// TwinCAT 3 PLC project Tc3_Event
// Title: Tc3_Event
// Company: www.peterzerlauth.com
// Author: Peter Zerlauth
// ProjectVersion: 0.0.0.7
// Description: Tc3_Event – TwinCAT 3 Event Logging Framework Copyright (c) Peter Zerlauth This component is provided under a Dual Licensing Model: 1. GPLv3 Open-Source License - Free for personal, educational, and non-commercial use. - Commercial use allowed only if the entire application is published under GPLv3, including all modifications to this code. - Requires full disclosure of source code for derivative works. 2. Commercial License - Required for integration into proprietary or closed-source products. - Removes all GPLv3 copyleft obligations. - Includes optional warranty, professional support, and long-term maintenance options. For commercial licensing, contact: info@peterzerlauth.com By using this Function Block you agree to the terms of the selected license.
// ProgramVersion: 3.1.4026.20
// libraries:
//   SysDir, * (System)
//   SysFile, * (System)
//   Tc2_Standard, * (Beckhoff Automation GmbH)
//   Tc2_System, * (Beckhoff Automation GmbH)
//   Tc2_Utilities, * (Beckhoff Automation GmbH)
//   Tc3_EventLogger, * (Beckhoff Automation GmbH)
//   Tc3_Module, * (Beckhoff Automation GmbH)
// project tree:
//   Argument/ FB_Argument.TcPOU (not stored), I_Argument.TcIO (not stored)
//   Event/ I_Event.TcIO, FB_Event.TcPOU
//   Global Variables/ GVL.TcGVL (not stored)
//   Helpers/File/ E_FileState.TcDUT (not stored), FB_File.TcPOU (not stored), I_File.TcIO (not stored)
//   Helpers/ F_Filter.TcPOU (not stored), F_Hash.TcPOU (not stored), F_InstancePath.TcPOU (not stored), F_Log.TcPOU (not stored), F_Print.TcPOU (not stored), F_Remove.TcPOU (not stored), LogLevel_To_Severity.TcPOU (not stored)
//   Logger/ E_LogLevel.TcDUT (not stored), I_Logger.TcIO (not stored)
//   Logger/FileLogger/ FB_FileLogger.TcPOU (not stored)
//   Logger/HmiLogger/ FB_HmiLogger.TcPOU (not stored)
//   Logger/Manager/ FB_LoggerManager.TcPOU (not stored)
//   Logger/TcLogger/ FB_TcLogger.TcPOU (not stored)
//   Message/ FB_Message.TcPOU (not stored)
//   Project Information/ F_GetCompany.TcPOU (not stored), F_GetTitle.TcPOU (not stored), F_GetVersion.TcPOU
//   Version/ Global_Version.TcGVL
// (motion and I/O tree: see PLC project plc01)
// real-time tasks:
//   TASK SlowTask: cycle T#20ms, priority 20, ADS port 350
//   TASK FastTask: cycle T#1ms, priority 1, ADS port 351

// ---- Version/Global_Version.TcGVL
{attribute 'TcGenerated'}
{attribute 'no-analysis'}
{attribute 'linkalways'}
// This function has been automatically generated from the project information.
VAR_GLOBAL CONSTANT
	{attribute 'const_non_replaced'}
	stLibVersion_Tc3_Event : ST_LibVersion := (iMajor := 0, iMinor := 0, iBuild := 0, iRevision := 7, nFlags := 0, sVersion := '0.0.0.7');
END_VAR

// ---- Event/I_Event.TcIO
INTERFACE I_Event

METHOD PUBLIC M_Critical : BOOL
VAR_INPUT
	sMessage:			STRING(255);
	nID:				UDINT;
END_VAR
END_METHOD

METHOD PUBLIC M_Error : BOOL
VAR_INPUT
	sMessage:			STRING(255);
	nID:				UDINT;
END_VAR
END_METHOD

METHOD PUBLIC M_Info : BOOL
VAR_INPUT
	sMessage:			STRING(255);
	nID:				UDINT;
END_VAR
END_METHOD

METHOD M_Reset : BOOL
VAR_INPUT
END_VAR
END_METHOD

METHOD PUBLIC M_Verbose : BOOL
VAR_INPUT
	sMessage:			STRING(255);
END_VAR
END_METHOD

METHOD PUBLIC M_Warning : BOOL
VAR_INPUT
	sMessage:			STRING(255);
	nID:				UDINT;
END_VAR
END_METHOD

PROPERTY PUBLIC P_Argument : I_Argument
GET
END_GET
END_PROPERTY

PROPERTY PUBLIC P_Logger : I_Logger
GET
END_GET
SET
END_SET
END_PROPERTY

END_INTERFACE

// ---- Event/FB_Event.TcPOU

{attribute 'reflection'} 
// Providing the event logger
FUNCTION_BLOCK FB_Event IMPLEMENTS I_Event
VAR_INPUT
	iLogger:					I_Logger;		// Interface has to be attached to a Valid target
END_VAR
VAR
    {attribute 'hide'} 
    {attribute 'instance-path'} 
    {attribute 'noinit'} 
    sInstancePath:				STRING(255);
	fbSymbolInfo: 				PLC_ReadSymInfoByNameEx;
	fbSystemTime: 				FB_LocalSystemTime;
	fbArguments:				FB_Argument;	
	fbVerbose:					FB_Message;
	fbInfo:						FB_Message;
	fbWarning:					FB_Message;
	fbError:					FB_Message;
	fbCritical:					FB_Message;
END_VAR
VAR_STAT
	nCycleTime:					UDINT;
	nTimestamp:					Tc2_Utilities.T_FILETIME64;		
END_VAR
(*
    Tc3_Event – TwinCAT 3 Event Logging Framework
    Copyright (c) Peter Zerlauth

    This component is provided under a Dual Licensing Model:

    1. GPLv3 Open-Source License
       - Free for personal, educational, and non-commercial use.
       - Commercial use allowed only if the entire application is published
         under GPLv3, including all modifications to this code.
       - Requires full disclosure of source code for derivative works.

    2. Commercial License
       - Required for integration into proprietary or closed-source products.
       - Removes all GPLv3 copyleft obligations.
       - Includes optional warranty, professional support, and long-term
         maintenance options.

    For commercial licensing, contact:
        info@peterzerlauth.com

    By using this Function Block you agree to the terms of the selected license.
*)

fbSymbolInfo();
IF nCycleTime <> TwinCAT_SystemInfoVarList._TaskInfo[GETCURTASKINDEXEX()].CycleTime THEN
	nCycleTime:= TwinCAT_SystemInfoVarList._TaskInfo[GETCURTASKINDEXEX()].CycleTime;
	fbSystemTime();
	nTimestamp:= SYSTEMTIME_TO_FILETIME64(fbSystemTime.systemTime);
	GVL.nTimestamp:= nTimestamp;	
END_IF

//FB_Init is always available implicitly and it is used primarily for initialization.
//The return value is not evaluated. For a specific influence, you can also declare the
//methods explicitly and provide additional code there with the standard initialization
//code. You can evaluate the return value.
METHOD FB_Init: BOOL
VAR_INPUT
    bInitRetains: BOOL; // TRUE: the retain variables are initialized (reset warm / reset cold)
    bInCopyCode: BOOL:= TRUE;  // TRUE: the instance will be copied to the copy code afterward (online change)   
END_VAR
fbSymbolInfo.SYMNAME:= F_InstancePath(sInstancePath);
fbSymbolInfo.PORT:= TwinCAT_SystemInfoVarList._AppInfo.AdsPort;
fbSymbolInfo.START:= TRUE;
fbSystemTime.bEnable:= TRUE;
END_METHOD

METHOD PUBLIC M_Critical : BOOL
VAR_INPUT
	sMessage:			STRING(255);
	nID:				UDINT;
END_VAR
VAR
	sArgument:			STRING;
	nPosition: 			INT;
END_VAR
IF sMessage = '' THEN
	RETURN;
END_IF

fbCritical.bActive:= TRUE;
fbCritical.sMessage:= sMessage;
fbCritical.eLogLevel:= E_LogLevel.Critical;
IF nID = 0 THEN
	fbCritical.nID:= F_Hash(sMessage);
ELSE
	fbCritical.nID:= nID;
END_IF
fbCritical.nTimestamp:= SYSTEMTIME_TO_FILETIME64(fbSystemTime.systemTime);
fbCritical.sArguments:= fbArguments.P_Value;
fbCritical.sDefault:= F_Print(sMessage, fbArguments.P_Value);
fbCritical.sSource:= fbSymbolInfo.SYMNAME;
fbCritical.sType:= fbSymbolInfo.SYMINFO.symDataType;

IF iLogger = 0 THEN
	F_Log(fbCritical);
ELSE
	iLogger.M_Log(fbCritical);
END_IF

	
fbArguments.M_Clear();
END_METHOD

METHOD PUBLIC M_Error : BOOL
VAR_INPUT
	sMessage:			STRING(255);
	nID:				UDINT;
END_VAR
VAR
	sArgument:			STRING;
	nPosition: 			INT;
END_VAR
IF sMessage = '' THEN
	RETURN;
END_IF

fbError.bActive:= TRUE;
fbError.sMessage:= sMessage;
fbError.eLogLevel:= E_LogLevel.Error;
IF nID = 0 THEN
	fbError.nID:= F_Hash(sMessage);
ELSE
	fbError.nID:= nID;
END_IF
fbError.nTimestamp:= SYSTEMTIME_TO_FILETIME64(fbSystemTime.systemTime);
fbError.sArguments:= fbArguments.P_Value;
fbError.sDefault:= F_Print(sMessage, fbArguments.P_Value);
fbError.sSource:= fbSymbolInfo.SYMNAME;
fbError.sType:= fbSymbolInfo.SYMINFO.symDataType;

IF iLogger = 0 THEN
	F_Log(fbError);
ELSE
	iLogger.M_Log(fbError);
END_IF

fbArguments.M_Clear();
END_METHOD

METHOD PUBLIC M_Info : BOOL
VAR_INPUT
	sMessage:			STRING(255);
	nID:				UDINT;
END_VAR
VAR
	sArgument:			STRING;
	nPosition: 			INT;
END_VAR
IF sMessage = '' THEN
	RETURN;
END_IF

fbInfo.bActive:= TRUE;
fbInfo.sMessage:= sMessage;
fbInfo.eLogLevel:= E_LogLevel.Info;
IF nID = 0 THEN
	fbInfo.nID:= F_Hash(sMessage);
ELSE
	fbInfo.nID:= nID;
END_IF
fbInfo.nTimestamp:= SYSTEMTIME_TO_FILETIME64(fbSystemTime.systemTime);
fbInfo.sArguments:= fbArguments.P_Value;
fbInfo.sDefault:= F_Print(sMessage, fbArguments.P_Value);
fbInfo.sSource:= fbSymbolInfo.SYMNAME;
fbInfo.sType:= fbSymbolInfo.SYMINFO.symDataType;

IF iLogger = 0 THEN
	F_Log(fbInfo);
ELSE
	iLogger.M_Log(fbInfo);
END_IF

fbArguments.M_Clear();
END_METHOD

METHOD M_Reset : BOOL
VAR_INPUT
END_VAR
VAR
	fbReset:					FB_Message;
END_VAR
fbReset.bActive:= TRUE;
fbReset.sMessage:= '###Reset###';
fbReset.eLogLevel:= E_LogLevel.Error;
fbReset.nID:= F_Hash(fbReset.sMessage);
fbReset.nTimestamp:= 0;
fbReset.sArguments:= '';
fbReset.sDefault:= '';
fbReset.sSource:= fbSymbolInfo.SYMNAME;
fbReset.sType:= fbSymbolInfo.SYMINFO.symDataType;

IF iLogger <> 0 THEN
	M_Reset:= iLogger.M_Log(fbReset);
END_IF
END_METHOD

METHOD PUBLIC M_Verbose : BOOL
VAR_INPUT
	sMessage:			STRING(255);		// content of the error message, placeholder %s
END_VAR
IF sMessage = '' THEN
	RETURN;
END_IF

fbVerbose.bActive:= TRUE;
fbVerbose.sMessage:= sMessage;
fbVerbose.eLogLevel:= E_LogLevel.Verbose;
fbVerbose.nID:= F_Hash(sMessage);
fbVerbose.nTimestamp:= SYSTEMTIME_TO_FILETIME64(fbSystemTime.systemTime);
fbVerbose.sArguments:= fbArguments.P_Value;
fbVerbose.sDefault:= F_Print(sMessage, fbArguments.P_Value);
fbVerbose.sSource:= fbSymbolInfo.SYMNAME;
fbVerbose.sType:= fbSymbolInfo.SYMINFO.symDataType;

IF iLogger = 0 THEN
	F_Log(fbVerbose);
ELSE
	iLogger.M_Log(fbVerbose);
END_IF


fbArguments.M_Clear();
END_METHOD

METHOD PUBLIC M_Warning : BOOL
VAR_INPUT
	sMessage:			STRING(255);
	nID:				UDINT;
END_VAR
IF sMessage = '' THEN
	RETURN;
END_IF

fbWarning.bActive:= TRUE;
fbWarning.sMessage:= sMessage;
fbWarning.eLogLevel:= E_LogLevel.Warning;
IF nID = 0 THEN
	fbWarning.nID:= F_Hash(sMessage);
ELSE
	fbWarning.nID:= nID;
END_IF
fbWarning.nTimestamp:= SYSTEMTIME_TO_FILETIME64(fbSystemTime.systemTime);
fbWarning.sArguments:= fbArguments.P_Value;
fbWarning.sDefault:= F_Print(sMessage, fbArguments.P_Value);
fbWarning.sSource:= fbSymbolInfo.SYMNAME;
fbWarning.sType:= fbSymbolInfo.SYMINFO.symDataType;

IF iLogger = 0 THEN
	F_Log(fbWarning);
ELSE
	iLogger.M_Log(fbWarning);
END_IF

fbArguments.M_Clear();
END_METHOD

PROPERTY PUBLIC P_Argument : I_Argument
GET
P_Argument:= fbArguments;
END_GET
END_PROPERTY

PROPERTY PUBLIC P_Logger : I_Logger
GET
P_Logger:= iLogger;
END_GET
SET
iLogger:= P_Logger;
END_SET
END_PROPERTY

END_FUNCTION_BLOCK

// ---- Project Information/F_GetVersion.TcPOU
// This function has been automatically generated from the project information.
{attribute 'signature_flag' := '1073741824'}
{attribute 'TcGenerated'}
{attribute 'no-analysis'}
FUNCTION F_GetVersion : ST_LibVersion
VAR_INPUT
	
END_VAR

F_GetVersion.iMajor := 0;
F_GetVersion.iMinor := 0;
F_GetVersion.iBuild := 0;
F_GetVersion.iRevision := 6;
F_GetVersion.sVersion := '0.0.0.6';
F_GetVersion.nFlags := 0;

END_FUNCTION
